{attribute 'qualified_only'}
{attribute 'strict'}
TYPE E_Joy :
(
	Joy_X,
	Joy_Y
);
END_TYPE

(* stored: Version 1.1.0.1, ProductVersion 3.1.4024.12
   DUT E_Joy: Id {2a2e134a-4acc-4965-b0c4-00f50e4983ec} *)
